INTERFACE ITF_BaseHMIComponent_Command EXTENDS ITF_BaseHMILoggerElement_Command

END_INTERFACE

(* stored: Version 1.1.0.1
   Itf ITF_BaseHMIComponent_Command: Id {5b79c555-bb4e-0612-21b2-9800599bdf7c} *)
